FUNCTION_BLOCK Lauflicht
VAR_INPUT
END_VAR
VAR_OUTPUT
END_VAR
VAR
	Blinker: TON;
	Zaehler : WORD;
END_VAR

Blinker(IN:= NOT Blinker.Q, PT:= T#100MS );

IF Blinker.Q THEN	Zaehler := Zaehler + 1;END_IF
IF Zaehler > 15 THEN Zaehler := 0;END_IF

DIO.DQW_1_16 := SHL(1 ,Zaehler);

END_FUNCTION_BLOCK

(* stored: Version 1.1.0.1, ProductVersion 3.1.4022.7
   POU Lauflicht: Id {7d16aa3e-6cbd-4e56-bda6-1c5f2746b937}, SpecialFunc None *)
